// TIA Portal project "Project3" (V16)

(* hardware
DEVICE "S7300/ET200M station_1"  S7-300 station
   slot 0: "Rail_0"  Rail  6ES7 390-1***0-0AA0
   slot 2: "PLC_1"  CPU 315-2 PN/DP  6ES7 315-2EH14-0AB0  V3.2
      slot 2: "PROFINET interface_1"  PN-IO
         slot 1: "Port_1"  Port
         slot 2: "Port_2"  Port
   slot 4: "DI 16x24VDC_1"  DI16 x 24VDC, interrupt  6ES7 321-7BH01-0AB0
   slot 5: "DI 16x24VDC_2"  DI16 x 24VDC, interrupt  6ES7 321-7BH01-0AB0
   slot 6: "DI 16x24VDC_3"  DI16 x 24VDC, interrupt  6ES7 321-7BH01-0AB0
   slot 7: "DO 16x24VDC/0.5A_1"  DO16 x 24VDC / 0.5A  6ES7 322-1BH01-0AA0
   slot 8: "DO 16x24VDC/0.5A_2"  DO16 x 24VDC / 0.5A  6ES7 322-1BH01-0AA0
   slot 9: "DO 16x24VDC/0.5A_3"  DO16 x 24VDC / 0.5A  6ES7 322-1BH01-0AA0
*)

// ===== PLC "PLC_1"  CPU 315-2 PN/DP =====

VAR_GLOBAL   // PLC tag table "Default tag table"
   "diEmerB" AT %I0.0 : Bool;
   "diPunchB" AT %I0.1 : Bool;
   "diGuardClosed" AT %I0.2 : Bool;
   "diPunchUp" AT %I0.3 : Bool;
   "diPunchDown" AT %I0.4 : Bool;
   "doPunch" AT %Q0.0 : Bool;
   "doSReadyIn" AT %Q0.1 : Bool;
   "doWReady" AT %Q0.2 : Bool;
   "doSGClosedIn" AT %Q0.3 : Bool;
   "doGuardDown" AT %Q0.4 : Bool;
   "mStart" AT %M100.0 : Bool;
   "mHelp1" AT %M200.1 : Bool;
   "mHelp2" AT %M200.2 : Bool;
   "Delay1" AT %T1 : Timer;
   "TV1" AT %QW66 : Word;
   "mHelp3" AT %M200.3 : Bool;
   "Delay3" AT %T3 : Timer;
   "mHelp4" AT %M200.4 : Bool;
   "mT3Elapsed" AT %M200.6 : Bool;
   "TV3" AT %QW68 : Word;
   "Delay2" AT %T2 : Timer;
   "mT2Elapsed" AT %M200.7 : Bool;
   "TV2" AT %QW70 : Word;
   "diStop" AT %I0.5 : Bool;
END_VAR

FUNCTION "fullAuto" : Void   // FC1, LAD
{ S7_Optimized_Access := 'FALSE' }
VERSION : 0.1
   VAR_TEMP   // added for the SCL form of the ladder/FBD networks
      _w1 : Bool;
      _w2 : Bool;
      _s5time1 : S5Time;
   END_VAR
BEGIN

REGION Network 1: Start machine
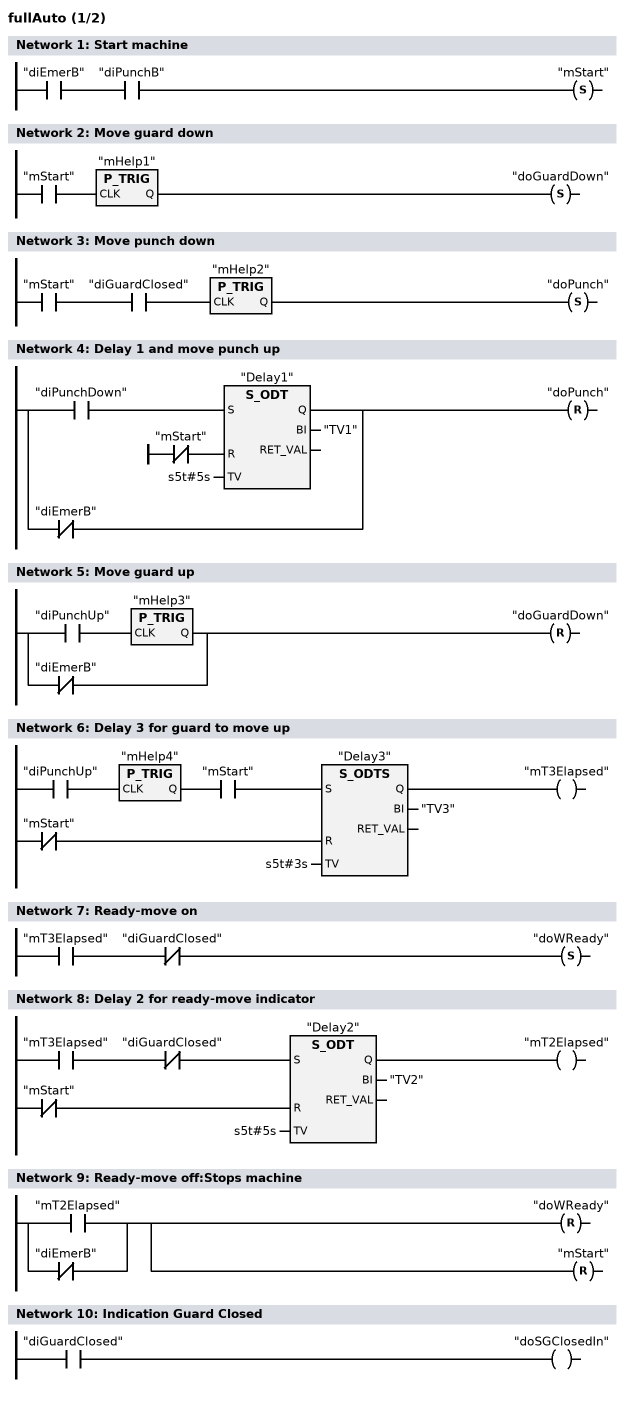
   RUNG wire#powerrail
      Contact( "diEmerB" )
      Contact( "diPunchB" )
      S_Coil( "mStart" )
   END_RUNG
   // the same network as SCL:
   IF "diEmerB" AND "diPunchB" THEN "mStart" := TRUE; END_IF;
END_REGION

REGION Network 2: Move guard down
   RUNG wire#powerrail
      Contact( "mStart" )
      P_Trig( "mHelp1" )
      S_Coil( "doGuardDown" )
   END_RUNG
   // the same network as SCL:
   #_w1 := "mStart" AND NOT "mHelp1";   // rising edge
   "mHelp1" := "mStart";
   IF #_w1 THEN "doGuardDown" := TRUE; END_IF;
END_REGION

REGION Network 3: Move punch down
   RUNG wire#powerrail
      Contact( "mStart" )
      Contact( "diGuardClosed" )
      P_Trig( "mHelp2" )
      S_Coil( "doPunch" )
   END_RUNG
   // the same network as SCL:
   #_w1 := "mStart" AND "diGuardClosed";
   #_w2 := #_w1 AND NOT "mHelp2";   // rising edge
   "mHelp2" := #_w1;
   IF #_w2 THEN "doPunch" := TRUE; END_IF;
END_REGION

REGION Network 4: Delay 1 and move punch up
   RUNG wire#powerrail
      Contact( "diPunchDown" )
      S_ODT(T_NO := "Delay1", R := wire#w1, TV := s5t#5s, BI => "TV1", RET_VAL =>)
      wire#w2
      R_Coil( "doPunch" )
   END_RUNG
   RUNG wire#powerrail
      I_Contact( "mStart" )
   END_RUNG wire#w1
   RUNG wire#powerrail
      I_Contact( "diEmerB" )
   END_RUNG wire#w2
   // the same network as SCL:
   #_s5time1 := S_ODT(T_NO := "Delay1",
                      S := "diPunchDown",
                      R := NOT "mStart",
                      TV := s5t#5s,
                      Q => #_w1,
                      BI => "TV1");
   IF #_w1 OR NOT "diEmerB" THEN "doPunch" := FALSE; END_IF;
END_REGION

REGION Network 5: Move guard up
   RUNG wire#powerrail
      Contact( "diPunchUp" )
      P_Trig( "mHelp3" )
      wire#w1
      R_Coil( "doGuardDown" )
   END_RUNG
   RUNG wire#powerrail
      I_Contact( "diEmerB" )
   END_RUNG wire#w1
   // the same network as SCL:
   #_w1 := "diPunchUp" AND NOT "mHelp3";   // rising edge
   "mHelp3" := "diPunchUp";
   IF #_w1 OR NOT "diEmerB" THEN "doGuardDown" := FALSE; END_IF;
END_REGION

REGION Network 6: Delay 3 for guard to move up
   RUNG wire#powerrail
      Contact( "diPunchUp" )
      P_Trig( "mHelp4" )
      Contact( "mStart" )
      S_ODTS(T_NO := "Delay3", R := wire#w1, TV := s5t#3s, BI => "TV3", RET_VAL =>)
      Coil( "mT3Elapsed" )
   END_RUNG
   RUNG wire#powerrail
      I_Contact( "mStart" )
   END_RUNG wire#w1
   // the same network as SCL:
   #_w1 := "diPunchUp" AND NOT "mHelp4";   // rising edge
   "mHelp4" := "diPunchUp";
   #_s5time1 := S_ODTS(T_NO := "Delay3",
                       S := #_w1 AND "mStart",
                       R := NOT "mStart",
                       TV := s5t#3s,
                       Q => #_w2,
                       BI => "TV3");
   "mT3Elapsed" := #_w2;
END_REGION

REGION Network 7: Ready-move on
   RUNG wire#powerrail
      Contact( "mT3Elapsed" )
      I_Contact( "diGuardClosed" )
      S_Coil( "doWReady" )
   END_RUNG
   // the same network as SCL:
   IF "mT3Elapsed" AND NOT "diGuardClosed" THEN "doWReady" := TRUE; END_IF;
END_REGION

REGION Network 8: Delay 2 for ready-move indicator
   RUNG wire#powerrail
      Contact( "mT3Elapsed" )
      I_Contact( "diGuardClosed" )
      S_ODT(T_NO := "Delay2", R := wire#w1, TV := s5t#5s, BI => "TV2", RET_VAL =>)
      Coil( "mT2Elapsed" )
   END_RUNG
   RUNG wire#powerrail
      I_Contact( "mStart" )
   END_RUNG wire#w1
   // the same network as SCL:
   #_s5time1 := S_ODT(T_NO := "Delay2",
                      S := "mT3Elapsed" AND NOT "diGuardClosed",
                      R := NOT "mStart",
                      TV := s5t#5s,
                      Q => #_w1,
                      BI => "TV2");
   "mT2Elapsed" := #_w1;
END_REGION

REGION Network 9: Ready-move off:Stops machine
   RUNG wire#powerrail
      Contact( "mT2Elapsed" )
      wire#w1
      R_Coil( "doWReady" )
   END_RUNG
   RUNG wire#powerrail
      I_Contact( "diEmerB" )
   END_RUNG wire#w1
   RUNG wire#w1
      R_Coil( "mStart" )
   END_RUNG
   // the same network as SCL:
   IF "mT2Elapsed" OR NOT "diEmerB" THEN
       "doWReady" := FALSE;
       "mStart" := FALSE;
   END_IF;
END_REGION

REGION Network 10: Indication Guard Closed
   RUNG wire#powerrail
      Contact( "diGuardClosed" )
      Coil( "doSGClosedIn" )
   END_RUNG
   // the same network as SCL:
   "doSGClosedIn" := "diGuardClosed";
END_REGION

REGION Network 11: Indication Emergency Button (EB)
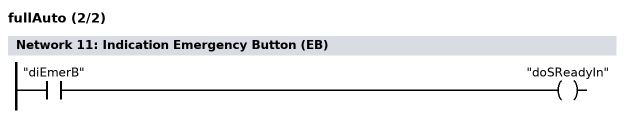
   RUNG wire#powerrail
      Contact( "diEmerB" )
      Coil( "doSReadyIn" )
   END_RUNG
   // the same network as SCL:
   "doSReadyIn" := "diEmerB";
END_REGION
END_FUNCTION

FUNCTION "semiAuto" : Void   // FC2, LAD
{ S7_Optimized_Access := 'FALSE' }
VERSION : 0.1
BEGIN

REGION Network 1: EmergencyButton(EB)
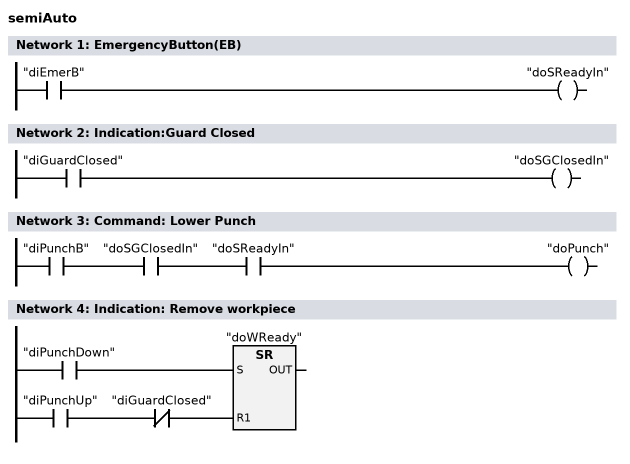
   RUNG wire#powerrail
      Contact( "diEmerB" )
      Coil( "doSReadyIn" )
   END_RUNG
   // the same network as SCL:
   "doSReadyIn" := "diEmerB";
END_REGION

REGION Network 2: Indication:Guard Closed
   RUNG wire#powerrail
      Contact( "diGuardClosed" )
      Coil( "doSGClosedIn" )
   END_RUNG
   // the same network as SCL:
   "doSGClosedIn" := "diGuardClosed";
END_REGION

REGION Network 3: Command: Lower Punch
   RUNG wire#powerrail
      Contact( "diPunchB" )
      Contact( "doSGClosedIn" )
      Contact( "doSReadyIn" )
      Coil( "doPunch" )
   END_RUNG
   // the same network as SCL:
   "doPunch" := "diPunchB" AND "doSGClosedIn" AND "doSReadyIn";
END_REGION

REGION Network 4: Indication: Remove workpiece
   RUNG wire#powerrail
      Contact( "diPunchDown" )
      S_SR(operand := "doWReady", r1 := wire#w1)
   END_RUNG
   RUNG wire#powerrail
      Contact( "diPunchUp" )
      I_Contact( "diGuardClosed" )
   END_RUNG wire#w1
   // the same network as SCL:
   IF "diPunchDown" THEN
       "doWReady" := TRUE;   // SR flip-flop
   END_IF;
   IF "diPunchUp" AND NOT "diGuardClosed" THEN "doWReady" := FALSE; END_IF;
END_REGION
END_FUNCTION

ORGANIZATION_BLOCK "Main"   // OB1, LAD
TITLE = "Main Program Sweep (Cycle)"
{ S7_Optimized_Access := 'FALSE' }
VERSION : 0.1
   VAR_TEMP
      OB1_EV_CLASS : Byte;   // Bits 0-3 = 1 (Coming event), Bits 4-7 = 1 (Event class 1)
      OB1_SCAN_1 : Byte;   // 1 (Cold restart scan 1 of OB 1), 3 (Scan 2-n of OB 1)
      OB1_PRIORITY : Byte;   // Priority of OB Execution
      OB1_OB_NUMBR : Byte;   // 1 (Organization block 1, OB1)
      OB1_RESERVED_1 : Byte;   // Reserved for system
      OB1_RESERVED_2 : Byte;   // Reserved for system
      OB1_PREV_CYCLE : Int;   // Cycle time of previous OB1 scan (milliseconds)
      OB1_MIN_CYCLE : Int;   // Minimum cycle time of OB1 (milliseconds)
      OB1_MAX_CYCLE : Int;   // Maximum cycle time of OB1 (milliseconds)
      OB1_DATE_TIME : Date_And_Time;   // Date and time OB1 started
   END_VAR
BEGIN

REGION Network 1
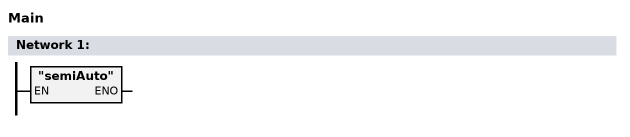
   RUNG wire#powerrail
      "semiAuto"()
   END_RUNG
   // the same network as SCL:
   "semiAuto"();
END_REGION
END_ORGANIZATION_BLOCK